TYPE TxHmiMru :
STRUCT
	status : DINT;
END_STRUCT
END_TYPE

(* stored: Version 1.1.0.1, ProductVersion 3.1.4020.12
   DUT TxHmiMru: Id {e7e539bd-33e9-404a-b164-57a9d3c3dbdc} *)
